SUBAPPLICATION Uebung_059_AX (* Reine Event-Schrittkette 8-Kanal (Adapter Version) *)
  (* Standard: 61499-2; Description: Copyright (c) 2026 Meisterschulen am Ostbahnhof This program and the accompanying materials are made available under the terms of the Eclipse Public License 2.0 which is available at https://www.eclipse.org/legal/epl-2.0/ SPDX-License-Identifier: EPL-2.0 *)
  (* Version 1.0, 2026-07-05, Franz Höpfinger, Meisterschulen am Ostbahnhof, generated solution *)
  PACKAGE Uebungen;
  IMPORT Uebungen::const::UT::DefaultPool::OutputNumber_N1;
  IMPORT logiBUS::io::DI::logiBUS_DI::Input_I1;
  IMPORT logiBUS::io::DI::logiBUS_DI::Input_I2;
  IMPORT logiBUS::io::DI::logiBUS_DI::Input_I3;
  IMPORT logiBUS::io::DI::logiBUS_DI::Input_I4;
  IMPORT logiBUS::io::DI::logiBUS_DI_Events::BUTTON_SINGLE_CLICK;
  IMPORT logiBUS::io::DQ::logiBUS_DO::Output_Q1;
  IMPORT logiBUS::io::DQ::logiBUS_DO::Output_Q2;
  IMPORT logiBUS::io::DQ::logiBUS_DO::Output_Q3;
  IMPORT logiBUS::io::DQ::logiBUS_DO::Output_Q4;
  IMPORT logiBUS::io::DQ::logiBUS_DO::Output_Q5;
  IMPORT logiBUS::io::DQ::logiBUS_DO::Output_Q6;
  IMPORT logiBUS::io::DQ::logiBUS_DO::Output_Q7;
  IMPORT logiBUS::io::DQ::logiBUS_DO::Output_Q8;
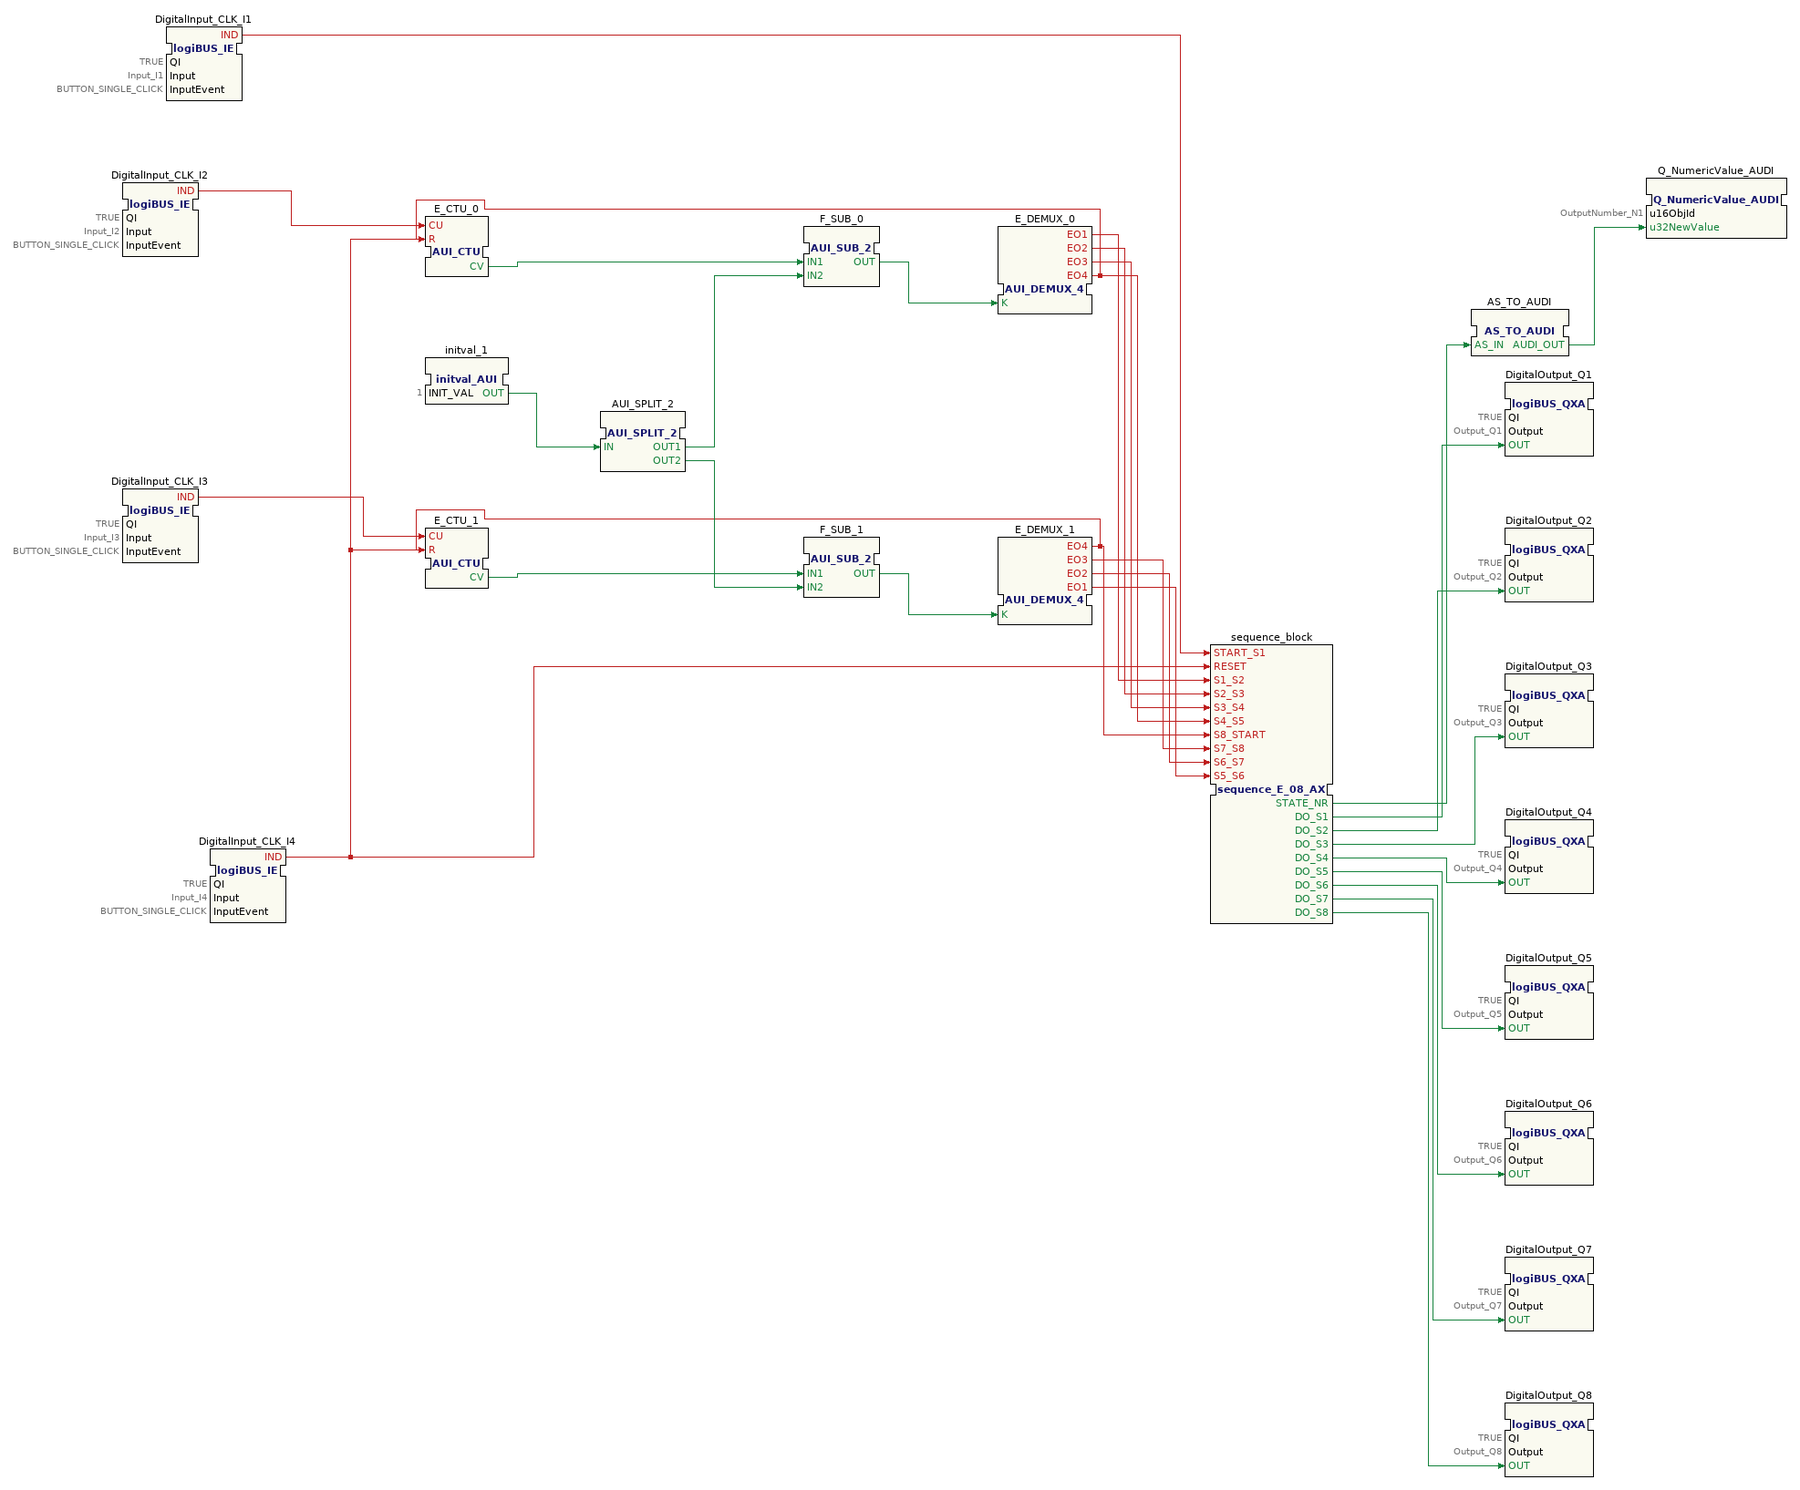
  FBS
    DigitalOutput_Q1 : logiBUS::io::DQ::logiBUS_QXA(QI := TRUE, Output := Output_Q1);
    DigitalOutput_Q2 : logiBUS::io::DQ::logiBUS_QXA(QI := TRUE, Output := Output_Q2);
    DigitalOutput_Q3 : logiBUS::io::DQ::logiBUS_QXA(QI := TRUE, Output := Output_Q3);
    DigitalOutput_Q4 : logiBUS::io::DQ::logiBUS_QXA(QI := TRUE, Output := Output_Q4);
    DigitalOutput_Q5 : logiBUS::io::DQ::logiBUS_QXA(QI := TRUE, Output := Output_Q5);
    DigitalOutput_Q6 : logiBUS::io::DQ::logiBUS_QXA(QI := TRUE, Output := Output_Q6);
    DigitalOutput_Q7 : logiBUS::io::DQ::logiBUS_QXA(QI := TRUE, Output := Output_Q7);
    DigitalOutput_Q8 : logiBUS::io::DQ::logiBUS_QXA(QI := TRUE, Output := Output_Q8);
    DigitalInput_CLK_I1 : logiBUS::io::DI::logiBUS_IE(QI := TRUE, Input := Input_I1, InputEvent := BUTTON_SINGLE_CLICK);
    E_CTU_0 : adapter::events::unidirectional::AUI_CTU;
    F_SUB_0 : adapter::iec61131::arithmetic::AUI_SUB_2;
    E_DEMUX_0 : adapter::events::unidirectional::AUI_DEMUX_4;
    DigitalInput_CLK_I2 : logiBUS::io::DI::logiBUS_IE(QI := TRUE, Input := Input_I2, InputEvent := BUTTON_SINGLE_CLICK);
    E_CTU_1 : adapter::events::unidirectional::AUI_CTU;
    F_SUB_1 : adapter::iec61131::arithmetic::AUI_SUB_2;
    E_DEMUX_1 : adapter::events::unidirectional::AUI_DEMUX_4;
    DigitalInput_CLK_I3 : logiBUS::io::DI::logiBUS_IE(QI := TRUE, Input := Input_I3, InputEvent := BUTTON_SINGLE_CLICK);
    DigitalInput_CLK_I4 : logiBUS::io::DI::logiBUS_IE(QI := TRUE, Input := Input_I4, InputEvent := BUTTON_SINGLE_CLICK);
    Q_NumericValue_AUDI : isobus::UT::Q::Q_NumericValue_AUDI(u16ObjId := OutputNumber_N1);
    AS_TO_AUDI : adapter::conversion::unidirectional::AS_TO_AUDI;
    sequence_block : logiBUS::utils::sequence::event::sequence_E_08_AX;
    initval_1 : adapter::types::unidirectional::AUI::initval::initval_AUI(INIT_VAL := 1);
    AUI_SPLIT_2 : adapter::events::unidirectional::AUI_SPLIT_2;
  END_FBS
  EVENT_CONNECTIONS
    DigitalInput_CLK_I1.IND TO sequence_block.START_S1;
    DigitalInput_CLK_I4.IND TO sequence_block.RESET;
    E_DEMUX_0.EO1 TO sequence_block.S1_S2;
    E_DEMUX_0.EO2 TO sequence_block.S2_S3;
    E_DEMUX_0.EO3 TO sequence_block.S3_S4;
    E_DEMUX_0.EO4 TO sequence_block.S4_S5;
    DigitalInput_CLK_I2.IND TO E_CTU_0.CU;
    DigitalInput_CLK_I3.IND TO E_CTU_1.CU;
    E_DEMUX_1.EO4 TO sequence_block.S8_START;
    E_DEMUX_1.EO3 TO sequence_block.S7_S8;
    E_DEMUX_1.EO2 TO sequence_block.S6_S7;
    E_DEMUX_1.EO1 TO sequence_block.S5_S6;
    DigitalInput_CLK_I4.IND TO E_CTU_1.R;
    DigitalInput_CLK_I4.IND TO E_CTU_0.R;
    E_DEMUX_0.EO4 TO E_CTU_0.R;
    E_DEMUX_1.EO4 TO E_CTU_1.R;
  END_CONNECTIONS
  ADAPTER_CONNECTIONS
    sequence_block.STATE_NR TO AS_TO_AUDI.AS_IN;
    AS_TO_AUDI.AUDI_OUT TO Q_NumericValue_AUDI.u32NewValue;
    sequence_block.DO_S1 TO DigitalOutput_Q1.OUT;
    sequence_block.DO_S2 TO DigitalOutput_Q2.OUT;
    sequence_block.DO_S3 TO DigitalOutput_Q3.OUT;
    sequence_block.DO_S4 TO DigitalOutput_Q4.OUT;
    sequence_block.DO_S5 TO DigitalOutput_Q5.OUT;
    sequence_block.DO_S6 TO DigitalOutput_Q6.OUT;
    sequence_block.DO_S7 TO DigitalOutput_Q7.OUT;
    sequence_block.DO_S8 TO DigitalOutput_Q8.OUT;
    E_CTU_0.CV TO F_SUB_0.IN1;
    AUI_SPLIT_2.OUT1 TO F_SUB_0.IN2;
    F_SUB_0.OUT TO E_DEMUX_0.K;
    E_CTU_1.CV TO F_SUB_1.IN1;
    AUI_SPLIT_2.OUT2 TO F_SUB_1.IN2;
    F_SUB_1.OUT TO E_DEMUX_1.K;
    initval_1.OUT TO AUI_SPLIT_2.IN;
  END_CONNECTIONS
END_SUBAPPLICATION
